// TIA Portal V19 export
VAR_GLOBAL   // PLC tag table "System"
   System_Byte AT %MB1 : Byte;
   FirstScan AT %M1.0 : Bool;
   DiagStatusUpdate AT %M1.1 : Bool;
   AlwaysTRUE AT %M1.2 : Bool;
   AlwaysFALSE AT %M1.3 : Bool;
   Clock_Byte AT %MB0 : Byte;
   Clock_10Hz AT %M0.0 : Bool;
   Clock_5Hz AT %M0.1 : Bool;
   "Clock_2.5Hz" AT %M0.2 : Bool;
   Clock_2Hz AT %M0.3 : Bool;
   "Clock_1.25Hz" AT %M0.4 : Bool;
   Clock_1Hz AT %M0.5 : Bool;
   "Clock_0.625Hz" AT %M0.6 : Bool;
   "Clock_0.5Hz" AT %M0.7 : Bool;
   ShuntTempSeb AT %M10.0 : Bool;
   ISS_PedestrialDoor AT %I508.3 : Bool;   // State Pedestral door acces control
   ISS_VacuumPumpRunning AT %I508.7 : Bool;   // State Vacuum pump runing, zero speed detection
END_VAR
